# EPICS IOC start-up script: test/startup/st.mcu010-SoftSlit-SimCfg.iocsh
epicsEnvSet("ECM_NUMAXES",     "6")
epicsEnvSet("MOTOR_PORT",      "$(SM_MOTOR_PORT=MCU1)")

epicsEnvSet("IPADDR",          "$(SM_IPADDR=192.168.242.60)")
epicsEnvSet("IPPORT",          "$(SM_IPPORT=48898)")
epicsEnvSet("AMSNETIDIOC",     "192.168.242.77.1.1")
epicsEnvSet("ASYN_PORT",       "$(SM_ASYN_PORT=MC_CPU1)")
epicsEnvSet("P",               "$(SM_P=IOC:)")
epicsEnvSet("R",               "")
epicsEnvSet("R",               "$(SM_R=m1)")
epicsEnvSet("AXIS_NO",         "$(SM_AXIS_NO=1)")
epicsEnvSet("DESC",            "$(SM_DESC=Lower=Right)")
epicsEnvSet("EGU",             "$(SM_EGU=mm)")
epicsEnvSet("PREC",            "$(SM_PREC=3)")
epicsEnvSet("SM_NOAXES",       "2")
# PILS would need this
#epicsEnvSet("ECM_OPTIONS",   "adsPort=852;amsNetIdRemote=192.168.88.60.1.1;amsNetIdLocal=$(AMSNETIDIOC)"
# But ADS needs this:
epicsEnvSet("ADSPORT",         852)
epicsEnvSet("REMOTEAMSNETID",  192.168.88.60.1.1)

# And this reads the input of an incremental encoder terminal
# on the EtherCAT bus. Works with the simulator.
# For real terminals the adresses must be adapted
epicsEnvSet("AXISCONFIG",      "stepSize=1.0;HomProc=1;HomPos=-66;cfgFile=./mcu010-SoftSlit-1.cfg;encoder=ADSPORT=501/.ADR.16#3040010,16#80000049,2,2")

< ethercatmcController.iocsh
< ethercatmcAxis.iocsh
< ethercatmcAxisdebug.iocsh

epicsEnvSet("AXISCONFIG",      "stepSize=1.0;HomProc=2;HomPos=61;cfgFile=./mcu010-SoftSlit-2.cfg;encoder=ADSPORT=501/.ADR.16#3040010,16#8000004F,2,2")

epicsEnvSet("R",               "$(SM_R=m2)")
epicsEnvSet("AXIS_NO",         "$(SM_AXIS_NO=2)")
epicsEnvSet("DESC",            "$(SM_DESC=Upper=Left)")
< ethercatmcAxis.iocsh
< ethercatmcAxisdebug.iocsh

## Logical axes and slit
epicsEnvSet("P",               "$(P)")
epicsEnvSet("SLIT",            "$(SM_SLIT=SltH-)")
epicsEnvSet("mXp",             "$(SM_mXp=m2)")
epicsEnvSet("mXn",             "$(SM_mXp=m1)")

## Slit
< ethercatmc2slit.iocsh
#########################
